// TwinCAT 3 PLC project B4Pipeline_Plc
// Title: B4Pipeline_Plc
// Company: Tc3 Project
// ProjectVersion: 1.0.0.0
// ProgramVersion: 3.1.4026.22
// libraries:
//   Tc2_Standard, * (Beckhoff Automation GmbH)
//   Tc2_System, * (Beckhoff Automation GmbH)
// project tree:
//   / PlcTask.TcTTO
//   POUs/ FB_PipelineInner.TcPOU, FB_PipelineStage.TcPOU, MAIN.TcPOU
// real-time tasks:
//   TASK PlcTask: cycle T#10ms, priority 20, ADS port 350

CONFIGURATION B4Pipeline_Plc
    RESOURCE PLC ON TwinCAT3
        TASK PlcTask(INTERVAL := T#10ms, PRIORITY := 20);
        PROGRAM MAIN WITH PlcTask : MAIN;
    END_RESOURCE
END_CONFIGURATION

// ---- POUs/MAIN.TcPOU
PROGRAM MAIN
VAR
END_VAR

END_PROGRAM

// ---- POUs/FB_PipelineInner.TcPOU
FUNCTION_BLOCK FB_PipelineInner
VAR_INPUT
    value : INT;
END_VAR
VAR_OUTPUT
    bError : BOOL;
END_VAR

// Inner raises an error for any negative input.
bError := value < 0;

END_FUNCTION_BLOCK

// ---- POUs/FB_PipelineStage.TcPOU
FUNCTION_BLOCK FB_PipelineStage
VAR_INPUT
    value : INT;
END_VAR
VAR_OUTPUT
    bError : BOOL;
END_VAR
VAR
    inner : FB_PipelineInner;
END_VAR

METHOD Step : INT
VAR
END_VAR
inner(value := value);
// MISSING: bError := inner.bError;
Step := value;
END_METHOD

END_FUNCTION_BLOCK
